(* PLC project  *)

CONFIGURATION StepIM_B
END_CONFIGURATION
